FUNCTION_BLOCK FB_Param_Add EXTENDS FB_BA_View
VAR
	TestAVal1			: FB_UDef_AVal				:= (iParent:=THIS^,		sDescription:='My user defined analog object',			eMode:=E_UDef_Mode.eAdd);
	TestAVal2			: FB_UDef_AVal				:= (iParent:=THIS^,		sDescription:='Another user defined analog object',		eMode:=E_UDef_Mode.eSubstract);
END_VAR
VAR
	{region 'Test'}
		nOffset			: UINT						:= 3;
	{endregion}
END_VAR

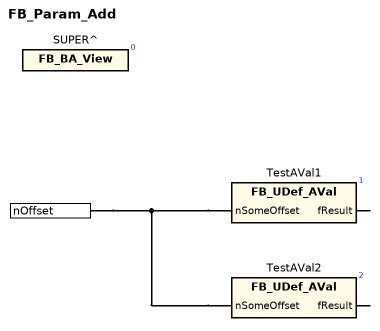
SUPER^(); // FB_BA_View
TestAVal1(nSomeOffset := nOffset); // FB_UDef_AVal
TestAVal2(nSomeOffset := nOffset); // FB_UDef_AVal

END_FUNCTION_BLOCK

(* stored: Version 1.1.0.1, ProductVersion 3.1.4024.9
   POU FB_Param_Add: Id {ee9c847e-86ab-4ab1-a8c8-e6dfc4e4d446}, SpecialFunc None *)
